                           //Temp OK, timers are done, the PS_ON can be turned on if there is no error.
                           IF (#TEMP_PSU_TEMP_REACHED = TRUE) AND
                               (#TEMP_ACTUAL_SETPOINT = 3) AND
                               (#ERROR_STAT = W#0) AND
                               (NOT #TEMP_Interlock) THEN

                               #TEMP_PSU_ON := TRUE;  //Heater can be turned ON
                               #TEMP_PSU_WARMUP := FALSE; //WarmUpOver
                               #TEMP_CurrentRampRate := 0.0;
                           END_IF;

                       ELSE
                           //ERROR: PSU can't be turned on because of an error
                           #ERRORS[15] := TRUE;
                           #TEMP_PSU_ON := FALSE;
                       END_IF;

                   END_IF;
               ELSE //ERROR if the PSU is in LOCAL mode
                   //Voltage limit adjust is not possible, Current adjus possible from 1% to 100% from the local potentiometer.
                   //ERROR: PSU can't operate from the PLC in LOCAL mode
                   #ERRORS[1] := TRUE;
                   #TEMP_PSU_STOPPED := TRUE;
                   #TEMP_PSU_ON := FALSE;
                   #TEMP_PSU_STARTED := FALSE;
                   #TEMP_PSU_WARMUP := FALSE;
                   #TEMP_PSU_TEMP_REACHED := FALSE;
                   #PSU_RSTAT.TOTAL_WARMUP_LEFT := 0;
                   #PSU_RSTAT.UPTIME_NO_HV := 0;
                   #PSU_RSTAT.WARMUP_LEFT_SP := 0;
                   #TEMP_ACTUAL_SETPOINT := 0;
                   #TEMP_CurrentRampRate := 0.0;
               END_IF;



               #TEMP_InterlockNeeded := FALSE;
               #TEMP_WarningNeeded := FALSE;

               //Interlock if PSU has internal fault
               IF (NOT #PSU_Inputs.FAULT) THEN
                   #TEMP_InterlockNeeded := TRUE;
                   //ERROR: PSU Interlock PSU has internal Fault
                   #ERRORS[10] := TRUE;
               END_IF;

               //Interlock handling during Warmup 
               #WARMUP_MONITOR(IN := ((#TEMP_IMON > (#TEMP_IPGM + #Temp_Tol_Warmup)) OR
                               (#TEMP_IMON < (#TEMP_IPGM - #Temp_Tol_Warmup))) AND
                               #TEMP_PSU_WARMUP,
                               PT := t#5s,
                               ET => #WARMUP_MONITOR_CurrTime,
                               Q => #WarmupMonitor_Tick);


               IF (#WarmupMonitor_Tick) THEN

                   #TEMP_InterlockNeeded := TRUE;
                   //ERROR: PSU Interlock during Warmup
                   #ERRORS[11] := TRUE;
                   #TEMP_InterlockNeeded := #TEMP_InterlockNeeded;
               END_IF;



                   //Check the Filament specific Current and Power maximum
                   IF (#TEMP_IMON > #MaxCurrentForFilament) OR (#TEMP_WMON > #MaxPowerForFilament) THEN
                       #TEMP_InterlockNeeded := TRUE;
                       //ERROR: PSU Interlock absolute maximum exeeded
                       #ERRORS[12] := TRUE;
                   END_IF;


                   //Interlocks for all status
                   IF (#TEMP_IMON > #PSU_RSTAT.I_HIHI) OR
                       (#TEMP_WMON > #PSU_RSTAT.W_HIHI) THEN
                       #TEMP_InterlockNeeded := TRUE;
                       //ERROR: PSU Interlock High limit exeeded
                       #ERRORS[13] := TRUE;
                   END_IF;

                   //Warning for all status
                   IF (#TEMP_IMON > #PSU_RSTAT.I_HIGH) OR
                       (#TEMP_WMON > #PSU_RSTAT.W_HIGH) THEN
                       #TEMP_WarningNeeded := TRUE;
                   END_IF;

                   //Interlock handling in all PSU status if it is Started
                   IF (#TEMP_PSU_STARTED) THEN

                       //Interlock and warning handling if PSU is ON and Blind_Out is passed
                       IF (#TEMP_PSU_ON AND #BlindOut_DONE) THEN
                           IF (#TEMP_IMON < #PSU_RSTAT.I_LOLO)
                               OR (#TEMP_WMON < #PSU_RSTAT.W_LOLO) THEN
                               #TEMP_InterlockNeeded := TRUE;
                               //ERROR: PSU Interlock Low limit exeeded
                               #ERRORS[14] := TRUE;
                           END_IF;

                           IF (#TEMP_IMON < #PSU_RSTAT.I_LOW)
                               OR (#TEMP_WMON < #PSU_RSTAT.W_LOW) THEN
                               #TEMP_WarningNeeded := TRUE;
                           END_IF;
                       END_IF;
                   END_IF;


               // Reset of the Interlock
               IF (NOT #TEMP_InterlockNeeded) THEN
                   // if Latching is OFF always empty the Interlock and warning bits
                   IF (#PSU_RSTAT.N_LATCH) THEN
                       #TEMP_Interlock := FALSE;
                       #TEMP_Warning := FALSE;
                       #PSU_RSTAT.IsFIRST := FALSE;

                   ELSE  // if Latching is ON empty the Interlock and warning bits only if RESET is applied 
                       IF (#TEMP_PSU_RESET) THEN
                           #TEMP_Interlock := FALSE;
                           #TEMP_Warning := FALSE;
                           #PSU_RSTAT.IsFIRST := FALSE;
                       END_IF;
                   END_IF;
               END_IF;

               //Apply the Interlock is needed
               IF #TEMP_InterlockNeeded THEN
                   #TEMP_Interlock := true;
               END_IF;

               //Apply the Interlock is needed
               IF #TEMP_WarningNeeded THEN
                   #TEMP_Warning := #TEMP_WarningNeeded;
               END_IF;

               //Blind out alarms after start for a given time
               #BlindOut(IN := #TEMP_PSU_ON,
                         PT := #AlarmBlindOutTime,
                         Q => #BlindOut_DONE);



               //Reaction to a Interlock
               IF (#TEMP_Interlock) THEN
                   IF (NOT #TimeStampUpdated) THEN
                       #ReadCLK_retval := RD_SYS_T(#PSU_RSTAT.TMPST);
                       #TimeStampUpdated := TRUE;
                   END_IF;
                   IF (#TEMP_IPGM <> 0.0) THEN
                       #IPGM_BeforeInterlock := #TEMP_IPGM; //Save it for debugging
                   END_IF;
                   #TEMP_PSU_STOPPED := TRUE;
                   #TEMP_PSU_ON := FALSE;
                   #TEMP_PSU_STARTED := FALSE;
                   #TEMP_PSU_WARMUP := FALSE;
                   #TEMP_ACTUAL_SETPOINT := 0;
                   #PSU_RSTAT.TOTAL_WARMUP_LEFT := 0;
                   #PSU_RSTAT.UPTIME_NO_HV := 0;
                   #PSU_RSTAT.WARMUP_LEFT_SP := 0;
                   #TEMP_CurrentRampRate := 0.0;

                   //Evaluate IsFirst
                   IF (#CPU_RCONF.INTERLOCK) THEN //SIM has already an Interlock
                       #PSU_RSTAT.IsFIRST := FALSE;
                   ELSE
                       #PSU_RSTAT.IsFIRST := TRUE;
                   END_IF;
               END_IF;

               //Set the SetPoint OUTPUT
               "PHYSICAL_TO_INT"(VAL => #PSU_Outputs.IPGM,
                                 EGU := #TEMP_IPGM,
                                 DTYP := "ENG_0-30A",
                                 ERROR => #I_SCALE_ERROR);

               IF (#I_SCALE_ERROR <> W#0) THEN
                   #ERRORS[5] := TRUE; //PSU IPGM SCALE Error
               END_IF;

               //Outputs
               #PSU_Outputs.ENA_IN := (#PSU_RSTAT.ON_STATUS OR #PSU_RSTAT.WARMUP) AND (NOT #TEMP_Interlock); // Turn on the Physical PSU 

               #PSU_Outputs.RESET := #TEMP_PSU_RESET;           //Apply reset to the PSU
               #PSU_Outputs.LOC_REM := TRUE;                      //SET always to REMOTE 
               #PSU_Outputs.VPGM := 0;                            //VPGM is not used for FILAMENT 

               //Copy TEMP variables to the RSTAT DB, so the values are SET only once! This way the EPICS flickering is avoided.
               #PSU_RSTAT.ON_STATUS := #TEMP_PSU_ON;
               #PSU_RSTAT.STARTED := #TEMP_PSU_STARTED;
               #PSU_RSTAT.STOPPED := #TEMP_PSU_STOPPED;
               #PSU_RSTAT.TEMP_REACHED := #TEMP_PSU_TEMP_REACHED;
               #PSU_RSTAT.WARMUP := #TEMP_PSU_WARMUP;
               #PSU_RSTAT.ACT_SP := INT_TO_REAL(#TEMP_ACTUAL_SETPOINT);
               //#PSU_RSTAT.INTERLOCK := #TEMP_Interlock;
               #PSU_RSTAT.WARNING := #TEMP_Warning;
               #PSU_RSTAT.I_RAMP_RATE := #TEMP_CurrentRampRate;
               //Other HMI visualisation
               IF (NOT #TEMP_Interlock) THEN // Freeze if there is an Interlock
                   #PSU_RSTAT.I_EGU_SP := #TEMP_IPGM;
               END_IF;

               //Return the ERROR word
               #PSU_RSTAT.ERR := #ERROR_STAT;

               IF (#ERROR_STAT <> 0) OR
                   (#TEMP_Interlock) THEN
                   #PSU_RSTAT.INTERLOCK := True;
               ELSE
                   #PSU_RSTAT.INTERLOCK := False;
               END_IF;

           END_IF;


   //Change LOG
   //v0.0 First implementation without warmup Setpoints
   //     - input simulation
   //     - cold and warm restart, different warmup time
   //    
   //v0.1 New functions:
   //     - implemented two warmup setpoint SP1 SP2 and SP3 for current during normal operation
   //     - cold and warm restart extended for three setpoint
   //     - implemented Ramping, can be turned on or off
   //     - tested with EPICS HMI
   //     - Low Pressure and High Pressure alarm and warning checking
   //     - NFORCE, NLATCH handling
   //     - IsFirst evaluation
   //     - extended error handling ErrorStatus word
   //
   //v0.2 New functions:
   //     - Added Change LOG and version header
   //     - High and low pressure automatic switchower using StateMachine ACT_STAT
   //     - Added Commands to the PSU_LOGIC input interface, so it can driven by the StateMachine added pulse generators
   //     - Fixed UptimeNOHV counter
   //    
   //v0.3 Fixed: time countdown is corrected from 0.1s basis to normal operation
   //     - New Intrelock Logik
   //     - Removed Low and High Pressure operation
   //     New functions: calculated total warmup for the StateMachine in Time format
   //    
   //v0.4 Fixed: 
   //     - Shorter variable names
   //     - Total time is now in S5TIME format
   //    
   //v0.5 Fixed: small visual changes
   //
   //v0.6 Fixed: Updated TOTAL_WARMUP_T calculation
   //     Tolarance for Warmup handling modified.
   //
   //v0.7 Fixed: Renaming variables V_SP I_SP 
   //     
   //v0.8 Fixed: Forcing bug for TEMP_IMON and TEMP_WMON 
   //     
   //v0.9 Fixed: SPs can be changed if the PS is ON but only after Warmup
   //     - Re-fix Total_warmup calculation, so the State machine will receive it before PSU_ON_CMD
   //v1.0 Fixed: Warning bit is also Latched now
   //
   //v1.1 Fixed: Changed the Data type for the set-points length.
   //     Integer type is not supported for more than 32 seconds (32767)
   //     - SP1_Length - INT -> DINT
   //     - SP1_Length - INT -> DINT
   //     - SP1_Length - INT -> DINT
   //     - The total length time requires at least +5 seconds to avoid a missmatch to the calculated
   //       time of the State Machine
   ////
   //TODO for the author: 
   //There is no reaction to the #PSU_RSTAT.PSU_UPTIME_NO_HV. Maybe a % dropoff will be necessary
END_FUNCTION_BLOCK

FUNCTION_BLOCK "SOLENOID_LOGIC"   // FB3002, SCL
{ S7_Optimized_Access := 'FALSE' }
VERSION : 0.1
   VAR_INPUT
      PSU_TYPE : Int;   // Power Supply Type ID
   END_VAR
   VAR_IN_OUT
      PSU_Outputs : "PSU_Outputs";   // General Output Signals from the PLC to the PSU
      PSU_Inputs : "PSU_Inputs";   // General Input Signals from the PSU to the PLC
      PSU_RSTAT : "SOLENOID_RST";   // PSU Status interface
      CPU_RCONF : "CPU_RCONF";   // SIM_GlobalData_Read
      CPU_WCONF : "CPU_WCONF";   // SIM_GlobalData_Write
      START_CMD : Bool;   // Start Command for StateMachine
      STOP_CMD : Bool;   // Stop Command for StateMachine
      PSU_WSTAT : "SOLENOID_WST";   // PSU Parameters interface
   END_VAR
   VAR
      ERROR_STAT : Word;   // Internal variable for ERROR bits
      ERRORS AT ERROR_STAT : Array[0..15] of Bool;   // Internal variable for ERROR bits
      BlindOut : TON_TIME;   // Blind out Limit checking
      PSU_UptimeNoHV : TON_TIME;   // Uptime timer in secs
      MaxCurrentForSolenoid : Real;   // The Maximum current for the filament defined by the supplier
      MaxVoltageForSolenoid : Real;   // The Maximum Power for the filament defined by the supplier
      AlarmBlindOutTime : Time;   // After turning on the PSU, the time till the limits supervisions are disabled
      BlindOut_DONE : Bool;   // Limits can be monitored now
      TEMP_IPGM : Real;   // Temp Current Output
      TEMP_IMON : Real;   // Temp Curernt Input
      TEMP_VMON : Real;   // Temp Voltage Input
      TEMP_PSU_ON : Bool;   // Temp variable for PSU_ON
      TEMP_PSU_STARTED : Bool;   // Temp variable for PSU_STARTED
      TEMP_PSU_STOPPED : Bool;   // Temp variable for PSU_STOPPED
      TEMP_PSU_RESET : Bool;   // Temp variable for PSU_RESET
      UptimeNoHV_TICK : Bool;   // Timer Tick bit
      V_SCALE_ERROR : Word;   // Scaling Error
      I_SCALE_ERROR : Word;   // Scaling Error
      TEMP_Interlock : Bool;
      TEMP_Warning : Bool;
      TEMP_InterlockNeeded : Bool;
      TEMP_WarningNeeded : Bool;
      PSU_STARTCMD_TP : TP_TIME;
      PSU_STARTCMD_TICK : Bool;
      PSU_RESETCMD_TP : TP_TIME;
      PSU_RESETCMD_TICK : Bool;
      PSU_STOPCMD_TP : TP_TIME;
      PSU_STOPCMD_TICK : Bool;
      PSU_STARTCMD_TP_WIRED : TP_TIME;
      PSU_STARTCMD_TICK_WIRED : Bool;
      PSU_STOPCMD_TP_WIRED : TP_TIME;
      PSU_STOPCMD_TICK_WIRED : Bool;
      VPGM_BeforeInterlock : Real;
      IPGM_BeforeInterlock : Real;
      TimeStampUpdated : Bool;
   END_VAR
   VAR_TEMP
      ReadCLK_retval : Int;
   END_VAR
BEGIN
   //Description: This SOLENOID_LOGIC FB handles Solenoid related tasks.
   //Author: Miklos Boros Tel:+36702072273 email:borosmiklos@gmail.com
   //Last update: 2016.12.05 11:00
   //Version: v0.4
   //Change log at the bottom of the code!

   //Error Bits description ***************************

           //Bit0;   EpicsBit8:  Initialisation error. No DTYP is given!
           //Bit1;   EpicsBit9:  PSU is in LOCAL mode. Set to REMOTE!
           //Bit2;   EpicsBit10: Analog Input IMON SCALE error!
           //Bit3;   EpicsBit11: Analog Input WMON SCALE error!
           //Bit4;   EpicsBit12: Analog Input VMON SCALE error!
           //Bit5;   EpicsBit13: Analog OutPut IPGM SCALE error!
           //Bit6;   EpicsBit14: 
           //Bit7;   EpicsBit15: 
           //Bit8;   EpicsBit0:  
           //Bit9;   EpicsBit1:  PSU SetPoint values are not in incresing order!
           //Bit10;  EpicsBit2:  Interlock PSU has internal faliure!
           //Bit11;  EpicsBit3:  Interlock absulute maximum for Current exeeded! 
           //Bit12;  EpicsBit4:  Interlock absulute maximum for Voltage exeeded!
           //Bit13;  EpicsBit5:  Interlock High limit exeeded while PSU_ON!
           //Bit14;  EpicsBit6:  Interlock Low limit exeeded while PSU_ON!
           //Bit15;  EpicsBit7:  PSU can't be turned on because of an error!


   //Init variables
   IF (NOT #TEMP_Interlock) THEN
       #ERROR_STAT := W#0; // Keep the value if an Iterlock happens
   END_IF;
   #TEMP_IPGM := 0.0;

   //First PLC Cícle
   IF (NOT #TEMP_PSU_STARTED) AND (NOT #TEMP_PSU_STOPPED) THEN
       #TEMP_PSU_STOPPED := TRUE;
   END_IF;


   //FEEDBACK SIGNALS **************************


   //IF (#PSU_WSTAT.WR_DATA) THEN

       //Feedback EPICS commands
       #PSU_RSTAT.FORCE_ON     := #PSU_WSTAT.FORCE;

       //Feedback Low Limits for Current and Voltage  
       #PSU_RSTAT.I_LOLO       := #PSU_WSTAT.I_LOLO;
       #PSU_RSTAT.I_LOW        := #PSU_WSTAT.I_LOW;
       #PSU_RSTAT.V_LOLO       := #PSU_WSTAT.V_LOLO;
       #PSU_RSTAT.V_LOW        := #PSU_WSTAT.V_LOW;

   //FORCE INPUT SIGNALS **************************
       //Feedback SIMULATION values
       #PSU_RSTAT.S_ON_STATUS    := #PSU_WSTAT.S_ON_STATUS;
       #PSU_RSTAT.S_IMON         := #PSU_WSTAT.S_IMON;
       #PSU_RSTAT.S_VMON         := #PSU_WSTAT.S_VMON;

       IF (#PSU_WSTAT.FORCE) THEN // If the FORCE in the HMI is pressed
           #PSU_RSTAT.FORCE_ON := #PSU_WSTAT.FORCE;
           IF (#PSU_RSTAT.N_FORCE = FALSE) THEN //Simulation of the values if NFORCE allows it

               //Take all the Simulated values from EPICS
               #PSU_Inputs.ON_STATUS := #PSU_WSTAT.S_ON_STATUS;
               #PSU_RSTAT.IMON := #PSU_WSTAT.S_IMON;
               #PSU_RSTAT.VMON := #PSU_WSTAT.S_VMON;
               //#CPU_RCONF.FORCE_DIS_MODE_ACT := TRUE;
           END_IF;
       END_IF;

       //Feedback the Intelock High limits with check
       IF (#PSU_WSTAT.I_HIHI < #MaxCurrentForSolenoid) THEN
           #PSU_RSTAT.I_HIHI := #PSU_WSTAT.I_HIHI;
       ELSE
           #PSU_RSTAT.I_HIHI := #MaxCurrentForSolenoid;
       END_IF;
       IF (#PSU_WSTAT.I_HIGH < #MaxCurrentForSolenoid) THEN
           #PSU_RSTAT.I_HIGH := #PSU_WSTAT.I_HIGH;
       ELSE
           #PSU_RSTAT.I_HIGH := #MaxCurrentForSolenoid;
       END_IF;
       IF (#PSU_WSTAT.V_HIHI < #MaxVoltageForSolenoid) THEN
           #PSU_RSTAT.V_HIHI := #PSU_WSTAT.V_HIHI;
       ELSE
           #PSU_RSTAT.V_HIHI := #MaxVoltageForSolenoid;
       END_IF;
       IF (#PSU_WSTAT.V_HIGH < #MaxVoltageForSolenoid) THEN
           #PSU_RSTAT.V_HIGH := #PSU_WSTAT.V_HIGH;
       ELSE
           #PSU_RSTAT.V_HIGH := #MaxVoltageForSolenoid;
       END_IF;


       //Feedback the SP1 SP2 SP3 currents with check
       IF (#PSU_WSTAT.I_SP < #MaxCurrentForSolenoid) THEN
           #PSU_RSTAT.I_SP := #PSU_WSTAT.I_SP;
       ELSE
           #PSU_RSTAT.I_SP := #MaxCurrentForSolenoid;
       END_IF;

       #PSU_WSTAT.WR_DATA := FALSE;

   //END_IF;

   IF (#PSU_RSTAT.FORCE_ON AND NOT #PSU_RSTAT.N_FORCE) THEN
       #CPU_RCONF.FORCE_DIS_MODE_ACT := TRUE;
   END_IF;


       //First PLC Cícle
       IF (NOT #TEMP_PSU_STARTED) AND (NOT #TEMP_PSU_STOPPED) THEN
           #TEMP_PSU_STOPPED := TRUE;
       END_IF;


       // PSU START COMMAND
       // If the PSU block receives the Start CMD the PSU_STARTED will be SET
       // #PSU_STARTCMD_TP(IN:=(#PSU_WSTAT.START), //Pulse generation for START_CMD coming from EPICS 
       //                  PT:=t#2s,
       //                  Q => #PSU_STARTCMD_TICK);
       #PSU_STARTCMD_TP_WIRED(IN := (#START_CMD),       //Pulse generation for START_CMD coming from StateMachine
                        PT := t#2s,
                        Q => #PSU_STARTCMD_TICK_WIRED);
       IF (#PSU_STARTCMD_TICK OR #PSU_STARTCMD_TICK_WIRED) AND (NOT #TEMP_Interlock) THEN
           #TEMP_PSU_STARTED := TRUE;
           #TEMP_PSU_STOPPED := FALSE;
       END_IF;
       IF (NOT #PSU_STARTCMD_TICK_WIRED) AND #START_CMD THEN
           #START_CMD := FALSE;
       END_IF;

       //PSU Reset COMMAND 
       #TEMP_PSU_RESET := FALSE; // the command is for 2s
       //#PSU_RESETCMD_TP(IN:=(#PSU_WSTAT.RESET OR #CPU_RCONF.RESET),
       #PSU_RESETCMD_TP(IN:= #CPU_RCONF.RESET,
                        PT:=t#2s
                        ,Q => #PSU_RESETCMD_TICK);

       IF (#PSU_RESETCMD_TICK) THEN
           #TEMP_PSU_RESET := TRUE;
       END_IF;

       // #PSU_STOPCMD_TP(IN:=(#PSU_WSTAT.STOP), //Pulse generation for STOP_CMD coming from EPICS
       //                 PT:=t#2s
       //                 ,Q=>#PSU_STOPCMD_TICK);

       #PSU_STOPCMD_TP_WIRED(IN := (#STOP_CMD),       //Pulse generation for STOP_CMD coming from StateMachine
                       PT := t#2s ,
                       Q => #PSU_STOPCMD_TICK_WIRED);

       //PSU STOP COMMAND 
      IF (#PSU_STOPCMD_TICK OR #PSU_STOPCMD_TICK_WIRED) THEN
           #TEMP_PSU_STOPPED            := TRUE;
           #TEMP_PSU_ON                 := FALSE;
           #TEMP_PSU_STARTED            := FALSE;
           #PSU_RSTAT.UPTIME_NO_HV      := 0;
       END_IF;
       IF (NOT #PSU_STOPCMD_TICK_WIRED) AND #STOP_CMD THEN
           #STOP_CMD := FALSE; 
       END_IF;


   IF (#PSU_TYPE = "PSU_NOT_DEFINED") THEN
           //Parametrization ERROR Type_Not_Filled_Out
           #ERRORS[0]                := TRUE;
           #TEMP_PSU_STOPPED         := TRUE;
           #TEMP_PSU_STARTED         := FALSE;
           #TEMP_PSU_ON              := FALSE;
           #PSU_RSTAT.UPTIME_NO_HV   := 0;
   END_IF;

   IF (#PSU_TYPE  = "PSU_KLYSTRON_SOLENOID") THEN //Type:Klystron FOCUS Solenoid

       #MaxCurrentForSolenoid := 16.0;  //Supplier specified Maximum Current (in Amp) 
       #MaxVoltageForSolenoid := 330.0; //Supplier specified Maximum Voltage (in Volt) 
       #AlarmBlindOutTime := t#2s; //The time before Interlock Low checking is enabled after PSU_ON

       //Feedback Max current and power to the HMI
       #PSU_RSTAT.SOL_MAX_I := #MaxCurrentForSolenoid;
       #PSU_RSTAT.SOL_MAX_V := #MaxVoltageForSolenoid;

       IF (NOT #PSU_RSTAT.FORCE_ON) OR (#PSU_RSTAT.N_FORCE = TRUE) THEN  //If PSU_FORCE is not applied, or disabled = normal operation          
           //Scale IMON 
           "INT_TO_PHYSICAL"(DTYP := "ENG_0-17A",
                             VAL := #PSU_Inputs.IMON,
                             EGU => #TEMP_IMON,
                             ERROR => #I_SCALE_ERROR);
           IF (#I_SCALE_ERROR <> W#0) THEN
               #ERRORS[2] := TRUE; //PSU IMON SCALE Error
           END_IF;
           #PSU_RSTAT.IMON := #TEMP_IMON;


           //Scale VMON
           "INT_TO_PHYSICAL"(DTYP := "ENG_0-300V",
                             VAL := #PSU_Inputs.VMON,
                             EGU => #TEMP_VMON,
                             ERROR => #V_SCALE_ERROR);
           IF (#V_SCALE_ERROR <> W#0) THEN
               #ERRORS[4] := TRUE; //PSU VMON SCALE Error
           END_IF;
           #PSU_RSTAT.VMON := #TEMP_VMON;

       END_IF;

       //Count PSU uptime without HV_ON in Secs Note: this is just an additional information, no action is done with this
       IF ((BYTE_TO_INT(#CPU_RCONF.ACT_STAT) < "STDBY")) AND (#TEMP_PSU_ON) THEN //StateMachine Status < 4 
           #PSU_UptimeNoHV(IN := NOT #UptimeNoHV_TICK,
                           PT := t#1s,
                           Q => #UptimeNoHV_TICK);
           IF (#UptimeNoHV_TICK) THEN
               #PSU_RSTAT.UPTIME_NO_HV := #PSU_RSTAT.UPTIME_NO_HV + 1;
           END_IF;
       ELSE
           #PSU_RSTAT.UPTIME_NO_HV := 0;
       END_IF;


       //Feedback the Intelock High limits with check
       // IF (#PSU_WSTAT.I_HIHI < #MaxCurrentForSolenoid) THEN
       //     #PSU_RSTAT.I_HIHI := #PSU_WSTAT.I_HIHI;
       // ELSE
       //     #PSU_RSTAT.I_HIHI := #MaxCurrentForSolenoid;
       // END_IF;
       // IF (#PSU_WSTAT.I_HIGH < #MaxCurrentForSolenoid) THEN
       //     #PSU_RSTAT.I_HIGH := #PSU_WSTAT.I_HIGH;
       // ELSE
       //     #PSU_RSTAT.I_HIGH := #MaxCurrentForSolenoid;
       // END_IF;
       // IF (#PSU_WSTAT.V_HIHI < #MaxVoltageForSolenoid) THEN
       //     #PSU_RSTAT.V_HIHI := #PSU_WSTAT.V_HIHI;
       // ELSE
       //     #PSU_RSTAT.V_HIHI := #MaxVoltageForSolenoid;
       // END_IF;
       // IF (#PSU_WSTAT.V_HIGH < #MaxVoltageForSolenoid) THEN
       //     #PSU_RSTAT.V_HIGH := #PSU_WSTAT.V_HIGH;
       // ELSE
       //     #PSU_RSTAT.V_HIGH := #MaxVoltageForSolenoid;
       // END_IF;


       // //Feedback the SP1 SP2 SP3 currents with check
       // IF (#PSU_WSTAT.I_SP < #MaxCurrentForSolenoid) THEN
       //     #PSU_RSTAT.I_SP := #PSU_WSTAT.I_SP;
       // ELSE
       //     #PSU_RSTAT.I_SP := #MaxCurrentForSolenoid;
       // END_IF;

       //Feedback Max current and power to the HMI
       #PSU_RSTAT.SOL_MAX_I := #MaxCurrentForSolenoid;
       #PSU_RSTAT.SOL_MAX_V := #MaxVoltageForSolenoid;

       //Blind out alarms after star for a given time
       #BlindOut(IN := #TEMP_PSU_ON,
                 PT := #AlarmBlindOutTime,
                 Q => #BlindOut_DONE);

       //CHECK the START conditions for PS_ON
           //1# START ENABE check
           IF (#TEMP_PSU_STARTED) AND (NOT #TEMP_Interlock) THEN
               IF (#ERROR_STAT = W#0) THEN

                   //Reset Timestamp refresh bit
                   #TimeStampUpdated := FALSE;

                   // TURN ON THE SOLENOID ********************
                   //Copy User SetPoint to the Output variable
                    #TEMP_IPGM := #PSU_RSTAT.I_SP;

                   //the PS_ON can be turned on if there is no error.
                    #TEMP_PSU_ON := TRUE;  //Heater can be turned ON

               ELSE
                   //ERROR: PSU can't be turned on because of an error
                   #ERRORS[15] := TRUE;
                   #TEMP_PSU_ON := FALSE;
               END_IF;

           END_IF;

   //        IF (NOT #PSU_RSTAT.N_LATCH) THEN
               #TEMP_InterlockNeeded := FALSE;
               #TEMP_WarningNeeded := FALSE;
   //        END_IF;

       //Interlock if PSU has internal fault
       IF ((NOT #PSU_Inputs.ON_STATUS) AND #BlindOut_DONE) THEN
           #TEMP_InterlockNeeded := TRUE;
           //ERROR: PSU Interlock PSU has internal Fault
           #ERRORS[10] := TRUE;
       END_IF;

           //Check the Solenoid specific Current and Power maximum
           IF (#TEMP_IMON > #MaxCurrentForSolenoid) THEN
               #TEMP_InterlockNeeded := TRUE;
               //ERROR: PSU Interlock absolute maximum for Current exeeded
               #ERRORS[11] := TRUE;
           END_IF;
           IF  (#TEMP_VMON > #MaxVoltageForSolenoid) THEN
               #TEMP_InterlockNeeded := TRUE;
               //ERROR: PSU Interlock absolute maximum for Voltage exeeded
               #ERRORS[12] := TRUE;
           END_IF;


           //Interlocks for all status
           IF (#TEMP_IMON > #PSU_RSTAT.I_HIHI) OR
               (#TEMP_VMON > #PSU_RSTAT.V_HIHI) THEN
               #TEMP_InterlockNeeded := TRUE;
               //ERROR: PSU Interlock High limit exeeded
               #PSU_Outputs.ENA_IN := False;
               #ERRORS[13] := TRUE;
           END_IF;

           //Warning for all status
           IF (#TEMP_IMON > #PSU_RSTAT.I_HIGH) OR
               (#TEMP_VMON > #PSU_RSTAT.V_HIGH) THEN
               #TEMP_WarningNeeded := TRUE;
           END_IF;


           //Interlock and warning handling for LOW limits if PSU is ON and Blind_Out is passed
           IF (#TEMP_PSU_ON AND #BlindOut_DONE) THEN
               IF (#TEMP_IMON < #PSU_RSTAT.I_LOLO)
                   OR (#TEMP_VMON < #PSU_RSTAT.V_LOLO) THEN
                   #TEMP_InterlockNeeded := TRUE;
                   //ERROR: PSU Interlock Low limit exeeded
                   #ERRORS[14] := TRUE;
               END_IF;

               IF (#TEMP_IMON < #PSU_RSTAT.I_LOW)
                   OR (#TEMP_VMON < #PSU_RSTAT.V_LOW) THEN
                   #TEMP_WarningNeeded := TRUE;
               END_IF;
           END_IF;


       // Reset of the Interlock
       IF (NOT #TEMP_InterlockNeeded) THEN
           // if Latching is OFF always empty the Interlock and warning bits
           IF (#PSU_RSTAT.N_LATCH) THEN
               #TEMP_Interlock := FALSE;
               #TEMP_Warning := FALSE;
               #PSU_RSTAT.IsFIRST := FALSE;
           ELSE  // if Latching is ON empty the Interlock and warning bits only if RESET is applied 
               IF (#TEMP_PSU_RESET) THEN
                   #TEMP_Interlock := FALSE;
                   #TEMP_Warning   := FALSE;
                   #PSU_RSTAT.IsFIRST := FALSE;
               END_IF;
           END_IF;
       END_IF;

       //Apply the Interlock if needed
       IF #TEMP_InterlockNeeded THEN
           #TEMP_Interlock := true;
       END_IF;

       //Apply the Warning if needed
       IF #TEMP_WarningNeeded THEN
           #TEMP_Warning := #TEMP_WarningNeeded;
       END_IF;



       //Reaction to a Interlock
       IF (#TEMP_Interlock) THEN
           IF (NOT #TimeStampUpdated) THEN
               #ReadCLK_retval := RD_SYS_T(#PSU_RSTAT.TMPST);
               #TimeStampUpdated := TRUE;
           END_IF;
           IF (#TEMP_IPGM <> 0.0) THEN
               #IPGM_BeforeInterlock := #TEMP_IPGM; //Save it for debugging
           END_IF;
           #TEMP_PSU_STOPPED := TRUE;
           #TEMP_PSU_ON      := FALSE;
           #TEMP_PSU_STARTED := FALSE;
           #PSU_RSTAT.UPTIME_NO_HV := 0;

           //Evaluate IsFirst
           IF (#CPU_RCONF.INTERLOCK) THEN //SIM has already an Interlock
               #PSU_RSTAT.IsFIRST := FALSE;
           ELSE
               #PSU_RSTAT.IsFIRST := TRUE;
           END_IF;
       END_IF;



       //Set the SetPoint OUTPUT
       "PHYSICAL_TO_INT"(VAL => #PSU_Outputs.IPGM,
                         EGU := #TEMP_IPGM,
                         DTYP := "ENG_0-17A",
                         ERROR => #I_SCALE_ERROR);

       IF (#I_SCALE_ERROR <> W#0) THEN
           #ERRORS[5] := TRUE; //PSU IPGM SCALE Error
       END_IF;



       //Outputs
       //#PSU_Outputs.ENA_IN := (#TEMP_PSU_ON) AND (NOT #TEMP_Interlock); // Turn on the Physical PSU
       #PSU_Outputs.LOC_REM := (#TEMP_PSU_ON) AND (NOT #TEMP_Interlock); // Turn on the Physical PSU

       //Copy TEMP variables to the RSTAT DB, so the values are SET only once! This way the EPICS flickering is avoided.
       #PSU_RSTAT.ON_STATUS := #TEMP_PSU_ON;
       #PSU_RSTAT.STARTED := #TEMP_PSU_STARTED;
       #PSU_RSTAT.STOPPED := #TEMP_PSU_STOPPED;
       #PSU_RSTAT.INTERLOCK := #TEMP_Interlock;
       #PSU_RSTAT.WARNING := #TEMP_Warning;

       //Other HMI visualisation
       IF (NOT #TEMP_Interlock) THEN // Freeze if there is an Interlock
           #PSU_RSTAT.I_EGU_SP := #TEMP_IPGM;
           #PSU_Outputs.ENA_IN := True;
       END_IF;

       //Return the ERROR word
       #PSU_RSTAT.ERR := #ERROR_STAT;



   END_IF;

   //Change LOG
   //v0.0 First implementation 
   //     - input simulation
   //    
   //v0.1 New functions:
   //     - Added first Solenoid LOGIC 
   //
   //v0.2 Updated logic:
   //     - Added first Solenoid LOGIC 
   //
   //v0.3 Updated logic:
   //     - Mojor update - testing with the SimBox 
   //
   //v0.4 Updated logic:
   //     Fixed warning bit latching 
   //

   //TODO for the author:
END_FUNCTION_BLOCK

FUNCTION "INT_S5TIME" : S5Time   // FC3000, STL
TITLE = Converts S5Time to Time in range 0..3276.7 seconds
{ S7_Optimized_Access := 'TRUE' }
VERSION : 0.1
// Function Converts Time in Integer [0..32767 ==> 0..3276.7seconds] to S5Time
// In case of Error ENO=False and 0 is returned
   VAR_INPUT
      I_TIME : Int;   // Time Value to be converted to S5Time
   END_VAR
   VAR_TEMP
      Time_Value : Int;   // Extracted Time Value [as Integer]
      Time_Base : Int;   // Extracted Time Base
   END_VAR
BEGIN

REGION Network 1: Select Time Base
         L     0;
         L     #I_TIME;  // Time as Integer 0..32767 --> 0..3276.7s
         <I;
         JC    CNVT;  // Jump to Convert if Time>=0
         CLR;  // Otherwise Clear ENO and finish
         SAVE;
         BE;

   CNVT: L     99;  // Limit for 10ms Time Base = 9.9seconds
         TAK;  // Toggle Accumulators to have Time in ACC1
         >=I;  // Time<=Limit?
         JC    T10m;  // Jump to 10ms Time Base
         L     999;  // Limit for 100ms Time Base = 99.9seconds [1m 39.9s.]
         TAK;
         >=I;  // Time<Limit?
         JC    T100;  // Jump to 100ms Time Base
         L     9999;  // Limit for 1s Time Base = 999seconds [16m 39s.]
         TAK;
         >=I;  // Time<=Limit?
         JC    T1s;  // Jump to 1s Time Base
         JU    T10s;  // Jump to 10s Time Base if Above
END_REGION

REGION Network 2
   T10m: L     10;  // Multiply int value times 10
         *I;  // to get time in 10ms units
         ITB;  // Convert to BCD. Time Base Bits are 00
         JU    ENDE;

   T100: ITB;  // Convert to BCD
         OW    W#16#1000;  // Apply Time Base [01 = 100ms]
         JU    ENDE;

   T1s:  L     10;  // Divide int value by 10
         /I;  // to get time in 1s units
         ITB;  // Convert to BCD.
         OW    W#16#2000;  // Apply Time Base [10 = 1s]
         JU    ENDE;

   T10s: L     100;  // Divide int value by 100
         /I;  // to get time in 10s units
         ITB;  // Convert to BCD.
         OW    W#16#3000;  // Apply Time Base [11 = 10s]
END_REGION

REGION Network 3: Issue Result and ENO=1
   ENDE: T     #INT_S5TIME;
         SET;
         SAVE;
END_REGION
END_FUNCTION